Universal Robots PolyScope program: bow_exp.urp

Program bow_exp (installation=string_planes directory=/programs createdIn=5.17.3 lastSavedIn=5.17.3 robotSerialNumber=20245501435)
Calibrated DH parameters: a=[0.000154, -0.137004, -0.385524, -0.00002, 0.000092, 0]; d=[0.162441, 211.794786, -230.585024, 18.923638, 0.099786, 0.09951]; alpha=[1.569493, -0.001902, 0.003874, 1.570111, -1.570167, 0]; deltaTheta=[0, -1.242934, 1.056292, 0.186646, 0.000002, 0.000001]
InitVariablesNode
Robot Program (runOnlyOnce=false)
  var_1 := 
  Call d_4
  var_1 := Waypoint_3
  Call a_2
  var_1 := Waypoint_2
SubProgram -> a_2
SubProgram -> d_4
SubProgram d_4 (keepSynchronizedWithDisk=false) programFile=/programs/d_4.urp
  MoveL speed 250 mm/s, acceleration 1200 mm/s^2 (useActiveTCP=true) feature=Plane_2
    Waypoint Variable (Variable): variable=var_1
    Waypoint Waypoint_3: TCP in base x=384.493 y=289.417 z=153.372 mm, rx=-1.5873 ry=-2.1561 rz=1.2208 rad; joints [-163.891, -53.511, 112.643, -101.372, -107.942, -172.933] deg; TCP offset x=28.21 y=-96.107 z=-99.69 mm, rx=0 ry=0 rz=0 rad; feature pose in base x=343.605 y=747.803 z=100.778 mm, rx=2.7685 ry=0.1285 rz=1.3673 rad
SubProgram a_2 (keepSynchronizedWithDisk=false) programFile=/programs/a_2.urp
  MoveL speed 250 mm/s, acceleration 1200 mm/s^2 (useActiveTCP=true) feature=Plane_1
    Waypoint Variable (Variable): variable=var_1
    Waypoint Waypoint_2 (Relative): relativeFromPosition TCP in base x=324.751 y=765.325 z=130.395 mm, rx=-1.4944 ry=-2.2779 rz=1.1569 rad; joints [-127.056, -14.743, 33.541, -62.029, -82.974, -153.445] deg; TCP in base x=480.541 y=452.328 z=220.562 mm, rx=-1.4944 ry=-2.2778 rz=1.1569 rad; joints [-152.229, -43.071, 77.058, -77.927, -101.277, -170.734] deg; feature pose in base x=325.716 y=793.387 z=118.207 mm, rx=-2.2082 ry=-0.2474 rz=-1.9195 rad
